INTERFACE I_JXCE1_StepperMotorControl

// Gets the controller state
PROPERTY ControllerState : E_JXCE1_State
GET
END_GET
END_PROPERTY

// Enables or disables the controller
PROPERTY Enable : BOOL
GET
END_GET
SET
END_SET
END_PROPERTY

// Gets or sets whether the axis is haleted
PROPERTY Hold : BOOL
GET
END_GET
SET
END_SET
END_PROPERTY

// Jogs backward with the defined speed
METHOD JogBwd
END_METHOD

// Jogs forward with the defined speed
METHOD JogFwd
END_METHOD

// Gets or sets the mode of operation for the unit
PROPERTY ModeOfOperation : E_JXCE1_ModeOfOperation
GET
END_GET
SET
END_SET
END_PROPERTY

// Gets or sets various movement data properties
PROPERTY MovementData : REFERENCE TO ST_JXCE1_MovementData
GET
END_GET
SET
END_SET
END_PROPERTY

// Moves to the target position with the defined speed. Returns TRUE when done
METHOD MoveToPosition : BOOL
VAR_INPUT
	speed		: REAL;
	position	: REAL;
END_VAR
VAR_OUTPUT
	error	: BOOL;	// If incorrect parameters are used, an error will be provided here
END_VAR
END_METHOD

// Resets the controller when called
METHOD Reset
END_METHOD

// Returns axis to origin
METHOD ReturnToOrigin
END_METHOD

// Gets the controller status structure
PROPERTY Status : REFERENCE TO ST_JXCE1_Status
GET
END_GET
END_PROPERTY

// Gets the stroke length (mm) of the actuator
PROPERTY StrokeLength : REAL
GET
END_GET
END_PROPERTY

END_INTERFACE

(* stored: Version 1.1.0.1, ProductVersion 3.1.4024.15
   Itf I_JXCE1_StepperMotorControl: Id {591e69f7-27c7-490e-b21c-1f8f935df247}
   Property ControllerState: Id {07112efa-ef21-0a40-35f4-e849001240cb}
   Get Get: Id {925e60bf-b482-0e00-1abb-5ef840831728}
   Property Enable: Id {c2e974ad-cf18-0125-2c21-5c488c8e84b9}
   Get Get: Id {da31aa66-e92f-078d-3ca9-e54450171d81}
   Set Set: Id {5ad5f2dc-0e73-0427-1498-86622c287d29}
   Property Hold: Id {d2e29514-bc5d-0805-28a6-349a7e0bf289}
   Get Get: Id {c52f095c-304d-01d5-1030-b3285a4cd1fa}
   Set Set: Id {14317072-6e80-01b0-1a0e-89cbfdce38c6}
   Method JogBwd: Id {f7b5f294-a10c-0e82-1569-5614cbaf881f}
   Method JogFwd: Id {688fd239-1930-028c-193b-bfb2c38229f8}
   Property ModeOfOperation: Id {da43743b-7869-0ceb-28b7-ee56c1e66df2}
   Get Get: Id {6aa3018d-bd07-0c84-2df3-f5885ee77c5c}
   Set Set: Id {32d16ece-5fdd-02dc-160a-531c5d109abb}
   Property MovementData: Id {e28ba497-29e0-0417-1ce4-0d1bde95843b}
   Get Get: Id {75a67e7f-88f2-0db9-0e3e-89b94534fb19}
   Set Set: Id {ee3ef076-2113-0a07-0daf-ff9613ffe5d0}
   Method MoveToPosition: Id {45e76dcc-c138-03b3-2b0e-2957adcac937}
   Method Reset: Id {9c29d6ae-36c1-0063-09b5-564afb349eb0}
   Method ReturnToOrigin: Id {3c9a5d29-c715-0cd6-2033-7d87c07c8f16}
   Property Status: Id {8a4ec173-3839-435d-9612-cc721b7c7729}
   Get Get: Id {99f94590-e258-4d90-bc59-eb5d73aa4a14}
   Property StrokeLength: Id {dd227f50-5e77-0a7d-3324-ebbc4306a3e5}
   Get Get: Id {cf8c7915-8da2-051b-3743-58645a89bb10} *)
